(* IEC 61131-3 sources: Lasal/CPU_5344_V01/Class/IFMSensor, 1 file *)

(* ---- IFMSensor.st ---- *)
(*!
<Class
	Name               = "IFMSensor"
	Revision           = "0.0"
	RealtimeTask       = "false"
	CyclicTask         = "true"
	DefCyclictime      = "10 ms"
	BackgroundTask     = "false"
	Sigmatek           = "false"
	OSInterface        = "false"
	HighPriority       = "false"
	Automatic          = "false"
	UpdateMode         = "Prescan"
	SharedCommandTable = "true"
	Objectsize         = "(284,120)">
	<Channels>
		<Server Name="ClassSvr" Visualized="false" Initialize="false" WriteProtected="true" Retentive="false"/>
		<Server Name="Dist" Visualized="false" Initialize="false" WriteProtected="true" Retentive="false"/>
		<Server Name="FcOn" Visualized="false" Initialize="false" WriteProtected="true" Retentive="false"/>
		<Server Name="Par_Multiply" Visualized="true" Initialize="true" WriteProtected="false" Retentive="SRam"/>
		<Server Name="Par_Offset" Visualized="true" Initialize="false" WriteProtected="false" Retentive="SRam"/>
		<Server Name="SetPoint" Visualized="false" Initialize="false" WriteProtected="false" Retentive="false"/>
		<Client Name="SDCI" Required="true" Internal="false"/>
		<Client Name="SDCIAsyncPara" Required="true" Internal="false"/>
	</Channels>
</Class>
*)
IFMSensor : CLASS
  //Servers:
	ClassSvr 	: SvrChCmd_DINT;
	FcOn 	: SvrCh_DINT;
	Dist 	: SvrCh_DINT;
	SetPoint 	: SvrCh_DINT;
	Par_Multiply 	: SvrCh_DINT;
	Par_Offset 	: SvrCh_DINT;
  //Clients:
	SDCI 	: CltChCmd_SDCIDevice;
	SDCIAsyncPara 	: CltChCmd_SDCIDevice_AsyncPara;
  //Variables:
		Data1 	: USINT;
		Data2 	: USINT;
		Data3 	: USINT;
		DAta 	: DINT;
  //Functions:

	FUNCTION VIRTUAL GLOBAL CyWork
		VAR_INPUT
			EAX 	: UDINT;
		END_VAR
		VAR_OUTPUT
			state (EAX) 	: UDINT;
		END_VAR;

	FUNCTION VIRTUAL GLOBAL SetPoint::Write
		VAR_INPUT
			input (EAX) 	: DINT;
		END_VAR
		VAR_OUTPUT
			result (EAX) 	: DINT;
		END_VAR;
  //Tables:
	FUNCTION @STD
		VAR_OUTPUT
			ret_code	: CONFSTATES;
		END_VAR;
	FUNCTION GLOBAL TAB @CT_;
END_CLASS;

#pragma usingLtd SDCIDevice
#pragma usingLtd SDCIDevice_AsyncPara

FUNCTION VIRTUAL GLOBAL IFMSensor::CyWork
	VAR_INPUT
		EAX 	: UDINT;
	END_VAR
	VAR_OUTPUT
		state (EAX) 	: UDINT;
	END_VAR

  Data := SDCI.GetReadPdoWord(ReadOffset:=0);
  FcOn := (Data AND 2#1) = 1;
  Dist := ((DATA/16) * Par_Multiply) + Par_Offset;
	state := READY;

END_FUNCTION

FUNCTION VIRTUAL GLOBAL IFMSensor::SetPoint::Write
	VAR_INPUT
		input (EAX) 	: DINT;
	END_VAR
	VAR_OUTPUT
		result (EAX) 	: DINT;
	END_VAR

	SetPoint := input;
  SDCIAsyncPara.ParaIndex.Write(input:=16#3c);
  SDCIAsyncPara.ParaSize.Write(input:=2);
  SDCIAsyncPara.ParaSubIndex.Write(input:=1);
  SDCIAsyncPara.ParaValue.Write(input:=SetPoint*256);
  SDCIAsyncPara.ParaRdWr.Write(input:=1);
	result := SetPoint;

END_FUNCTION
